// TIA Portal V17 export
// export: Created 2025-06-25T13:13:03.5445527Z, ExportSetting WithDefaults, DisplayName Totally Integrated Automation Portal, DisplayVersion V17 Update 8, DisplayName TIA Portal Openness, DisplayVersion V17 Update 8, DisplayName TIA Portal Version Control Interface, DisplayVersion V17, DisplayName STEP 7 Professional, DisplayVersion V17 Update 8, DisplayName STEP 7 Safety, DisplayVersion V17 Update 6, DisplayName WinCC Advanced, DisplayVersion V17 Update 8
FUNCTION "InitCurrentSettings" : Void   // FC29, FBD
TITLE = Load data from DB_StaticData
{ S7_Optimized_Access := 'TRUE' }
AUTHOR : Heaten
VERSION : 0.1
// stored: AutoNumber true, IsIECCheckEnabled false, SetENOAutomatically false, UDAEnableTagReadback false
   VAR_OUTPUT
      RetVal_Fluid : Int;
      RetVal_System : Int;
      RetValve_Compressor : Int;
      Busy : Bool;
   END_VAR
   VAR_TEMP
      Busy_Fluid : Bool;
      Busy_System : Bool;
      Busy_Compressor : Bool;
      "Counter" : Int;
      Trigger : Bool;
   END_VAR
BEGIN

REGION Network 1: Load fluid data
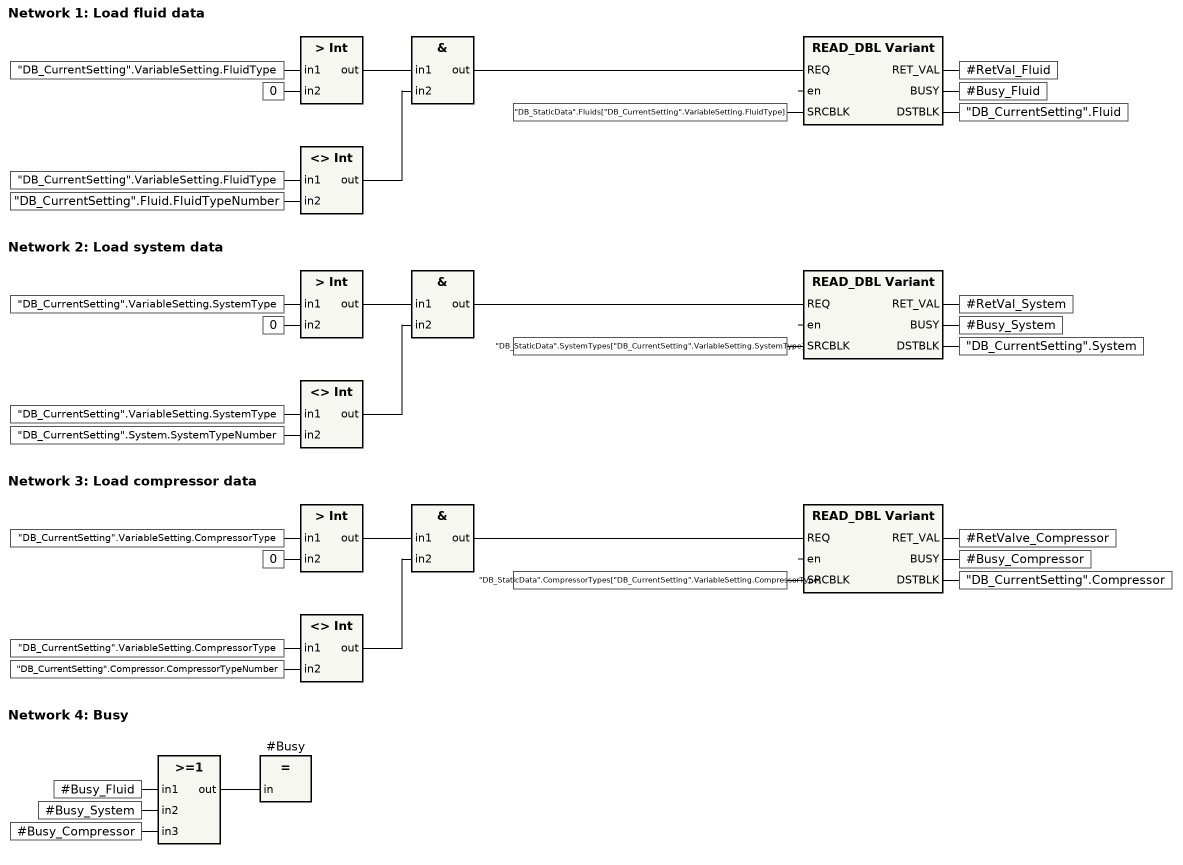
   #RetVal_Fluid := READ_DBL(REQ := ("DB_CurrentSetting".VariableSetting.FluidType > 0) AND ("DB_CurrentSetting".VariableSetting.FluidType <> "DB_CurrentSetting".Fluid.FluidTypeNumber),
                           SRCBLK := "DB_StaticData".Fluids["DB_CurrentSetting".VariableSetting.FluidType],
                           BUSY => #Busy_Fluid,
                           DSTBLK => "DB_CurrentSetting".Fluid);
END_REGION

REGION Network 2: Load system data
   #RetVal_System := READ_DBL(REQ := ("DB_CurrentSetting".VariableSetting.SystemType > 0) AND ("DB_CurrentSetting".VariableSetting.SystemType <> "DB_CurrentSetting".System.SystemTypeNumber),
                           SRCBLK := "DB_StaticData".SystemTypes["DB_CurrentSetting".VariableSetting.SystemType],
                           BUSY => #Busy_System,
                           DSTBLK => "DB_CurrentSetting".System);
END_REGION

REGION Network 3: Load compressor data
   #RetValve_Compressor := READ_DBL(REQ := ("DB_CurrentSetting".VariableSetting.CompressorType > 0) AND ("DB_CurrentSetting".VariableSetting.CompressorType <> "DB_CurrentSetting".Compressor.CompressorTypeNumber),
                           SRCBLK := "DB_StaticData".CompressorTypes["DB_CurrentSetting".VariableSetting.CompressorType],
                           BUSY => #Busy_Compressor,
                           DSTBLK => "DB_CurrentSetting".Compressor);
END_REGION

REGION Network 4: Busy
   #Busy := #Busy_Fluid OR #Busy_System OR #Busy_Compressor;
END_REGION
END_FUNCTION
